(* Logix 5000 project; controller test vendor 1 type 14 code 65 rev 20.19; software revision 20.04 *)

TASK MainTask (continuous, watchdog 500 ms) : AK47Detector, HallwaySensor, MapInputs

MODULES
   Controller : vendor 1 type 14 code 65 (CompactLogixL35Controller 0, rev 20.19)
      LocalENB : 1769-L35E Ethernet Port (CompactLogixL35Ethernet 1, rev 20.11)
      Local : CompactBus (CompactVirtualAdapter 3, rev 20.11)
         digital : vendor 1 type 7 code 66 (Compact 2, rev 1.1, Output RPI 20 ms)
         Analog : vendor 1 type 10 code 33 (Compact 1, rev 1.1, Output RPI 80 ms)
END_MODULES

VAR_GLOBAL   (* controller tags *)
   door_snsr_status : ALIAS FOR Local:2:I.Data.0;
   hallway_snsr_status : ALIAS FOR Local:2:I.Data.1;
   nerfgun_motor_on : ALIAS FOR Local:2:I.Data.3;
   nerfgun_position_fire : ALIAS FOR Local:2:I.Data.2;
END_VAR

PROGRAM AK47Detector   (* main routine Aa_Main *)
VAR
   app_trigger_motor : ALIAS FOR Local:2:I.Data.3;   // Input 3 Triggers Motor On or Off HIGH - ON LOW - OFF
   app_trigger_nerfgun_position : ALIAS FOR Local:2:I.Data.2;   // Input 2 Positions Nerf Gun HIGH - Position Fire LOW - Position Hide
   nerfgun_motor : ALIAS FOR Local:2:O.Data.3;   // Output 3 HIGH - On LOW - Off
   nerfgun_position : ALIAS FOR Local:2:O.Data.2;   // Output 2 HIGH - Nerfgun Down LOW - Pull Nerfgun Up
END_VAR

ROUTINE Aa_Main   (* ladder *)
// Out2
// - HIGH (Bring Gun Up)
// - LOW (Drop Gun Down)
// Out3
// - HIGH (Turn Motor On)
// - LOW (Turn Motor Off)
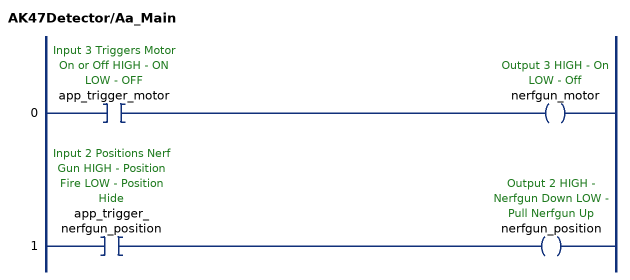
   0 (stored rung type 13): XIC(app_trigger_motor)OTE(nerfgun_motor);
   1 (stored rung type 13): XIC(app_trigger_nerfgun_position)OTE(nerfgun_position);
END_ROUTINE
END_PROGRAM

PROGRAM DoorSensor
VAR
   door_snsr_in : ALIAS FOR Local:2:I.Data.0;   // From front door sensor (yellow wire)
   door_snsr_out : ALIAS FOR Local:2:O.Data.0;
END_VAR

ROUTINE Ab_Main   (* ladder *)
// Routine for the front door sensor
   0 (stored rung type 13): ;
END_ROUTINE
END_PROGRAM

PROGRAM Faults
END_PROGRAM

PROGRAM HallwaySensor   (* main routine Ac_Main *)
VAR
   hallway_snsr_in : ALIAS FOR Local:2:I.Data.1;   // The white wire input from the Photo Eye sensor in the hallway.
END_VAR

ROUTINE Ac_Main   (* ladder *)
   0 (stored rung type 13): ;
END_ROUTINE
END_PROGRAM

PROGRAM MapInputs
VAR
   light : ALIAS FOR Local:2:O.Data.0;
   start_switch : ALIAS FOR Local:2:I.Data.0;   // test switch
END_VAR

ROUTINE MainRoutine   (* ladder *)
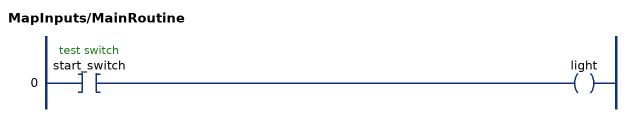
   0: XIC(start_switch)OTE(light);
END_ROUTINE
END_PROGRAM
